TYPE DUT_70x1CoeData :
STRUCT
     (* Hardware *)
    //Readbacks
    {attribute 'pytmc' := '
     pv: MAX:CUR
     io: i
     field: DESC Max Current
    '}
    nMaxCurrent : WORD;
    {attribute 'pytmc' := '
     pv: REDUC:CUR
     io: i
     field: DESC Reduced Current
    '}
    nReducedCurrent : WORD;
    {attribute 'pytmc' := '
     pv: NOM:VOL
     io: i
     field: DESC Nominal Voltage
    '}
    nNominalVoltage: WORD;
    {attribute 'pytmc' := '
     pv: MTR:STP
     io: i
     field: DESC Motor Fullsteps
    '}
    nMotorFullSteps: WORD;
    {attribute 'pytmc' := '
     pv: SPD:RNG
     io: i
     field: DESC Speed Range
    '}
    nSpeedRange: WORD;
END_STRUCT
END_TYPE

(* stored: Version 1.1.0.1, ProductVersion 3.1.4022.18
   DUT DUT_70x1CoeData: Id {482c096a-5d07-4231-a5de-180f2bbde26d} *)
